{attribute 'GeneratedUsingTerminal: ER1518-0002-0018'}
{attribute addProperty BoxType "ER1518-0002-0018"}
{attribute addProperty Id "InputAT %I*ARRAY[0..7] OF BOOL8"}
{attribute addProperty CRC "3697175534"}
{attribute addProperty Size "8"}
TYPE DIG_Inputs_CAFF6004 EXTENDS InputBase_8311D824 :
STRUCT
	{attribute addProperty Name "Input"}
	Input AT %I* : ARRAY[0..7] OF BOOL;
END_STRUCT
END_TYPE

(* stored: Version 1.2.0.0, ProductVersion 3.1.4024.11
   DUT DIG_Inputs_CAFF6004: Id {6f888048-0a94-432e-83a2-0768c3da496c} *)
